PROGRAM MAIN_SFC
VAR

END_VAR

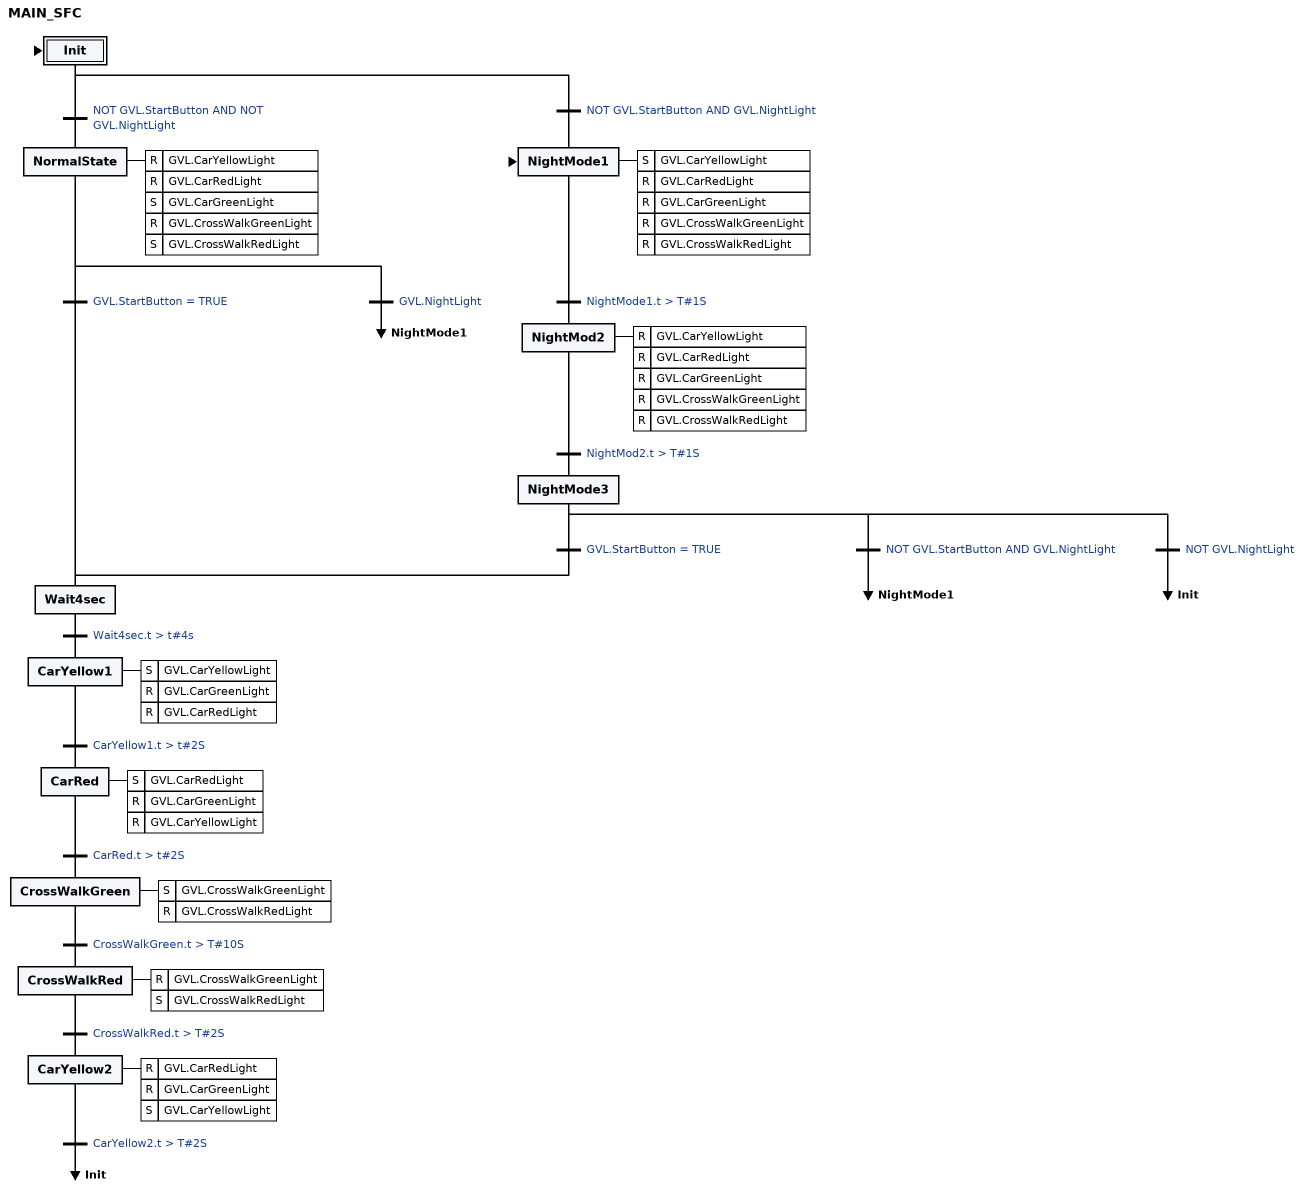
INITIAL_STEP Init:
END_STEP
TRANSITION FROM Init TO NormalState
    := NOT GVL.StartButton AND NOT GVL.NightLight;
END_TRANSITION
STEP NormalState:
    GVL.CarYellowLight(R);
    GVL.CarRedLight(R);
    GVL.CarGreenLight(S);
    GVL.CrossWalkGreenLight(R);
    GVL.CrossWalkRedLight(S);
END_STEP
TRANSITION FROM NormalState TO Wait4sec
    := GVL.StartButton = TRUE;
END_TRANSITION
TRANSITION FROM NormalState TO NightMode1
    := GVL.NightLight;
END_TRANSITION
TRANSITION FROM Init TO NightMode1
    := NOT GVL.StartButton AND GVL.NightLight;
END_TRANSITION
STEP NightMode1:
    GVL.CarYellowLight(S);
    GVL.CarRedLight(R);
    GVL.CarGreenLight(R);
    GVL.CrossWalkGreenLight(R);
    GVL.CrossWalkRedLight(R);
END_STEP
TRANSITION FROM NightMode1 TO NightMod2
    := NightMode1.t > T#1S;
END_TRANSITION
STEP NightMod2:
    GVL.CarYellowLight(R);
    GVL.CarRedLight(R);
    GVL.CarGreenLight(R);
    GVL.CrossWalkGreenLight(R);
    GVL.CrossWalkRedLight(R);
END_STEP
TRANSITION FROM NightMod2 TO NightMode3
    := NightMod2.t > T#1S;
END_TRANSITION
STEP NightMode3:
END_STEP
TRANSITION FROM NightMode3 TO Wait4sec
    := GVL.StartButton = TRUE;
END_TRANSITION
TRANSITION FROM NightMode3 TO NightMode1
    := NOT GVL.StartButton AND GVL.NightLight;
END_TRANSITION
TRANSITION FROM NightMode3 TO Init
    := NOT GVL.NightLight;
END_TRANSITION
STEP Wait4sec:
END_STEP
TRANSITION FROM Wait4sec TO CarYellow1
    := Wait4sec.t > t#4s;
END_TRANSITION
STEP CarYellow1:
    GVL.CarYellowLight(S);
    GVL.CarGreenLight(R);
    GVL.CarRedLight(R);
END_STEP
TRANSITION FROM CarYellow1 TO CarRed
    := CarYellow1.t > t#2S;
END_TRANSITION
STEP CarRed:
    GVL.CarRedLight(S);
    GVL.CarGreenLight(R);
    GVL.CarYellowLight(R);
END_STEP
TRANSITION FROM CarRed TO CrossWalkGreen
    := CarRed.t > t#2S;
END_TRANSITION
STEP CrossWalkGreen:
    GVL.CrossWalkGreenLight(S);
    GVL.CrossWalkRedLight(R);
END_STEP
TRANSITION FROM CrossWalkGreen TO CrossWalkRed
    := CrossWalkGreen.t > T#10S;
END_TRANSITION
STEP CrossWalkRed:
    GVL.CrossWalkGreenLight(R);
    GVL.CrossWalkRedLight(S);
END_STEP
TRANSITION FROM CrossWalkRed TO CarYellow2
    := CrossWalkRed.t > T#2S;
END_TRANSITION
STEP CarYellow2:
    GVL.CarRedLight(R);
    GVL.CarGreenLight(R);
    GVL.CarYellowLight(S);
END_STEP
TRANSITION FROM CarYellow2 TO Init
    := CarYellow2.t > T#2S;
END_TRANSITION

END_PROGRAM

(* stored: Version 1.1.0.1, ProductVersion 3.1.4024.15
   POU MAIN_SFC: Id {88118615-1af4-460c-889a-a44738ab5137}, SpecialFunc None *)
